// TIA Portal V17 export
// export: Created 2023-02-26T22:28:47.9107326Z, ExportSetting WithDefaults, DisplayName Totally Integrated Automation Portal, DisplayVersion V17, DisplayName TIA Portal Openness, DisplayVersion V17, DisplayName TIA Portal Version Control Interface, DisplayVersion V17, DisplayName TIA Portal Test Suite Advanced, DisplayVersion V17, DisplayName STEP 7 Professional, DisplayVersion V17, DisplayName SIMATIC Energy Suite, DisplayVersion V17, DisplayName STEP 7 Safety, DisplayVersion V17, DisplayName WinCC Professional, DisplayVersion V17
DATA_BLOCK "ERR_ChangeMode_DB"   // DB23
VERSION : 0.1
// stored: AutoNumber true, InstanceOfName ERR_ChangeMode, InstanceOfType FB
"ERR_ChangeMode"
   // VAR_INPUT
   //    StartLine : Bool;
   //    StopLine : Bool;
   //    ModeAuto : Bool;
   //    ModeManual : Bool;
   //    ResetButton : Bool;
   //    AlarmSiren : Bool;
   //    FirstScan : Bool;
   // END_VAR
   // VAR_OUTPUT
   //    Error : Bool;
   // END_VAR
   // VAR
   //    S1 : Bool;
   //    S2 : Bool;
   //    S3 : Bool;
   //    S4 : Bool;
   //    S5 : Bool;
   //    P_ResetButton : Bool;
   // END_VAR
BEGIN
END_DATA_BLOCK
